// TIA Portal project "ejercicio1" (V15.1)

(* hardware
DEVICE "HMI_1"  KTP700 Basic PN
   slot 0: "HMI_1"  KTP700 Basic PN  6AV2 123-2GB03-0AX0  15.1.0.0
   slot 1: "HMI_RT_1"  KTP700 Basic PN  6AV2 123-2GB03-0AX0  15.1.0.0
   slot 5: "HMI_1.IE_CP_1"  PROFINET Interface  15.0.1.0
      slot 1: "Interfaz PROFINET_1"  PROFINET Interface
         slot 1: "Port_1"  Port
DEVICE "S7-1200 station_1"  S7-1200 Station
   slot 0: "Rack_0"  S7-1200 Rack  Rack  V1.0
   slot 1: "PLC_1"  CPU 1215C AC/DC/Rly  6ES7 215-1BG40-0XB0  V4.2
*)

// ===== PLC "PLC_1"  CPU 1215C AC/DC/Rly =====

VAR_GLOBAL   // PLC tag table "Tabla de variables estándar"
   "q1" AT %M0.0 : Bool;   // estado 1
   "q2" AT %M0.1 : Bool;   // estado 2
   "q3" AT %M0.2 : Bool;   // estado 3
   "q4" AT %M0.3 : Bool;   // estado 4
   "q5" AT %M0.4 : Bool;   // estado 5
   "q6" AT %M0.5 : Bool;   // estado 6
   "MP1" AT %M1.0 : Bool;   // mover der-iz
   "MP2" AT %M1.1 : Bool;   // mover iz-der
   "XV" AT %M1.2 : Bool;   // electrovalvula
   "MC" AT %M1.3 : Bool;   // rodillos
   "MV" AT %M1.4 : Bool;   // ventilador
   "M" AT %M2.0 : Bool;   // boton encendido
   "S1" AT %M2.1 : Bool;   // final de carrera iz
   "S2" AT %M2.2 : Bool;   // final de carrera der
   "S3" AT %M2.3 : Bool;   // detector de coches
   "P" AT %M2.4 : Bool;   // boton paro
END_VAR

ORGANIZATION_BLOCK "Main"   // OB1, LAD, ProgramCycle
TITLE = "Main Program Sweep (Cycle)"
{ S7_Optimized_Access := 'TRUE' }
VERSION : 0.1
   VAR_INPUT
      Initial_Call : Bool;   // Initial call of this OB
      Remanence : Bool;   // =True, if remanent data are available
   END_VAR
BEGIN

REGION Network 1: estado 6: paro
   // si detectamos el boton de paro reseteamos todo y activamos el motor para que regrese a su posicion original
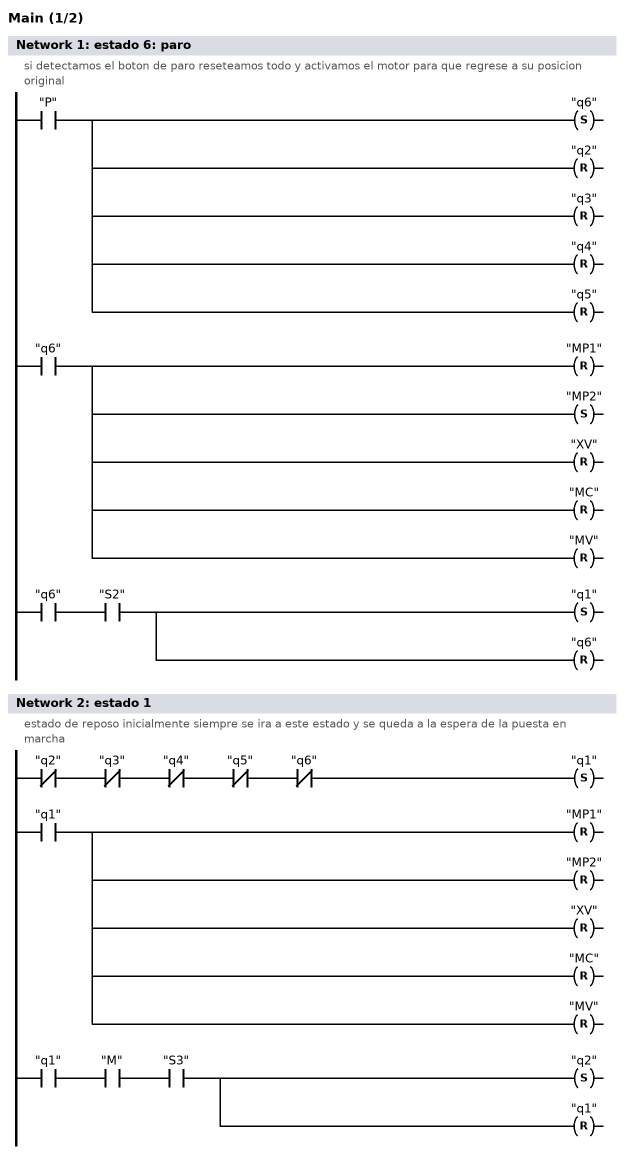
   RUNG wire#powerrail
      Contact( "P" )
      wire#w1
      S_Coil( "q6" )
   END_RUNG
   RUNG wire#w1
      R_Coil( "q2" )
   END_RUNG
   RUNG wire#w1
      R_Coil( "q3" )
   END_RUNG
   RUNG wire#w1
      R_Coil( "q4" )
   END_RUNG
   RUNG wire#w1
      R_Coil( "q5" )
   END_RUNG
   RUNG wire#powerrail
      Contact( "q6" )
      wire#w2
      R_Coil( "MP1" )
   END_RUNG
   RUNG wire#w2
      S_Coil( "MP2" )
   END_RUNG
   RUNG wire#w2
      R_Coil( "XV" )
   END_RUNG
   RUNG wire#w2
      R_Coil( "MC" )
   END_RUNG
   RUNG wire#w2
      R_Coil( "MV" )
   END_RUNG
   RUNG wire#powerrail
      Contact( "q6" )
      Contact( "S2" )
      wire#w3
      S_Coil( "q1" )
   END_RUNG
   RUNG wire#w3
      R_Coil( "q6" )
   END_RUNG
   // the same network as SCL:
   IF "P" THEN
       "q6" := TRUE;
       "q2" := FALSE;
       "q3" := FALSE;
       "q4" := FALSE;
       "q5" := FALSE;
   END_IF;
   IF "q6" THEN
       "MP1" := FALSE;
       "MP2" := TRUE;
       "XV" := FALSE;
       "MC" := FALSE;
       "MV" := FALSE;
   END_IF;
   IF "q6" AND "S2" THEN
       "q1" := TRUE;
       "q6" := FALSE;
   END_IF;
END_REGION

REGION Network 2: estado 1
   // estado de reposo inicialmente siempre se ira a este estado y se queda a la espera de la puesta en marcha
   RUNG wire#powerrail
      I_Contact( "q2" )
      I_Contact( "q3" )
      I_Contact( "q4" )
      I_Contact( "q5" )
      I_Contact( "q6" )
      S_Coil( "q1" )
   END_RUNG
   RUNG wire#powerrail
      Contact( "q1" )
      wire#w1
      R_Coil( "MP1" )
   END_RUNG
   RUNG wire#w1
      R_Coil( "MP2" )
   END_RUNG
   RUNG wire#w1
      R_Coil( "XV" )
   END_RUNG
   RUNG wire#w1
      R_Coil( "MC" )
   END_RUNG
   RUNG wire#w1
      R_Coil( "MV" )
   END_RUNG
   RUNG wire#powerrail
      Contact( "q1" )
      Contact( "M" )
      Contact( "S3" )
      wire#w2
      S_Coil( "q2" )
   END_RUNG
   RUNG wire#w2
      R_Coil( "q1" )
   END_RUNG
   // the same network as SCL:
   IF NOT "q2" AND NOT "q3" AND NOT "q4" AND NOT "q5" AND NOT "q6" THEN "q1" := TRUE; END_IF;
   IF "q1" THEN
       "MP1" := FALSE;
       "MP2" := FALSE;
       "XV" := FALSE;
       "MC" := FALSE;
       "MV" := FALSE;
   END_IF;
   IF "q1" AND "M" AND "S3" THEN
       "q2" := TRUE;
       "q1" := FALSE;
   END_IF;
END_REGION

REGION Network 3: Estado 2
   // ida lavado
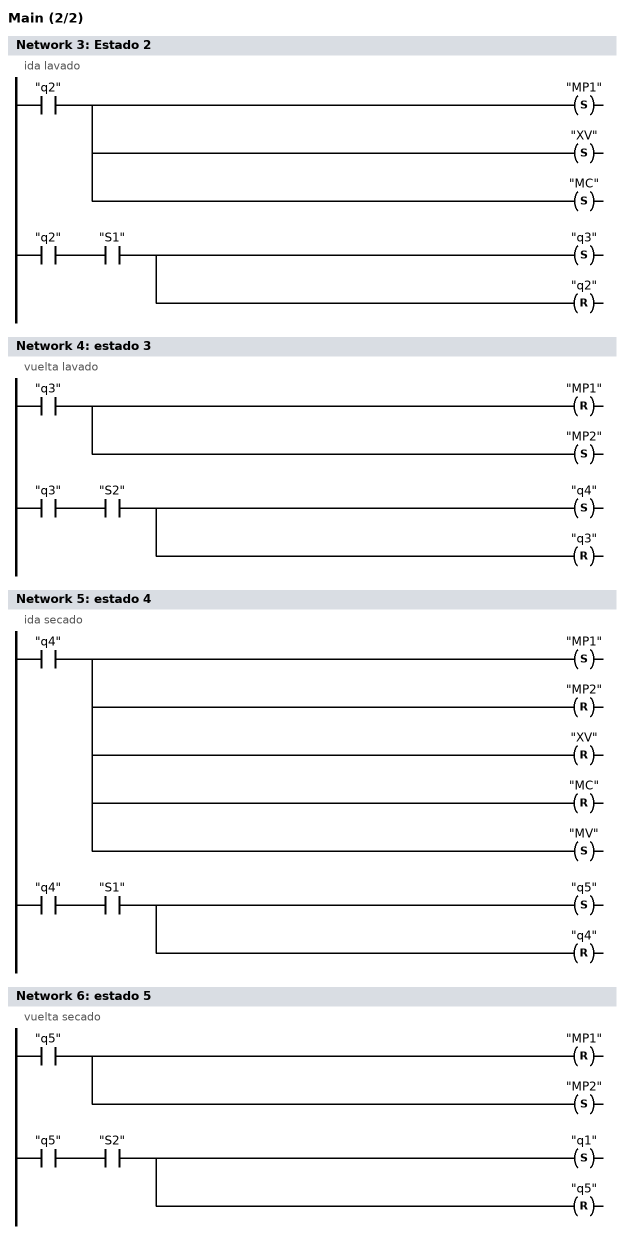
   RUNG wire#powerrail
      Contact( "q2" )
      wire#w1
      S_Coil( "MP1" )
   END_RUNG
   RUNG wire#w1
      S_Coil( "XV" )
   END_RUNG
   RUNG wire#w1
      S_Coil( "MC" )
   END_RUNG
   RUNG wire#powerrail
      Contact( "q2" )
      Contact( "S1" )
      wire#w2
      S_Coil( "q3" )
   END_RUNG
   RUNG wire#w2
      R_Coil( "q2" )
   END_RUNG
   // the same network as SCL:
   IF "q2" THEN
       "MP1" := TRUE;
       "XV" := TRUE;
       "MC" := TRUE;
   END_IF;
   IF "q2" AND "S1" THEN
       "q3" := TRUE;
       "q2" := FALSE;
   END_IF;
END_REGION

REGION Network 4: estado 3
   // vuelta lavado
   RUNG wire#powerrail
      Contact( "q3" )
      wire#w1
      R_Coil( "MP1" )
   END_RUNG
   RUNG wire#w1
      S_Coil( "MP2" )
   END_RUNG
   RUNG wire#powerrail
      Contact( "q3" )
      Contact( "S2" )
      wire#w2
      S_Coil( "q4" )
   END_RUNG
   RUNG wire#w2
      R_Coil( "q3" )
   END_RUNG
   // the same network as SCL:
   IF "q3" THEN
       "MP1" := FALSE;
       "MP2" := TRUE;
   END_IF;
   IF "q3" AND "S2" THEN
       "q4" := TRUE;
       "q3" := FALSE;
   END_IF;
END_REGION

REGION Network 5: estado 4
   // ida secado
   RUNG wire#powerrail
      Contact( "q4" )
      wire#w1
      S_Coil( "MP1" )
   END_RUNG
   RUNG wire#w1
      R_Coil( "MP2" )
   END_RUNG
   RUNG wire#w1
      R_Coil( "XV" )
   END_RUNG
   RUNG wire#w1
      R_Coil( "MC" )
   END_RUNG
   RUNG wire#w1
      S_Coil( "MV" )
   END_RUNG
   RUNG wire#powerrail
      Contact( "q4" )
      Contact( "S1" )
      wire#w2
      S_Coil( "q5" )
   END_RUNG
   RUNG wire#w2
      R_Coil( "q4" )
   END_RUNG
   // the same network as SCL:
   IF "q4" THEN
       "MP1" := TRUE;
       "MP2" := FALSE;
       "XV" := FALSE;
       "MC" := FALSE;
       "MV" := TRUE;
   END_IF;
   IF "q4" AND "S1" THEN
       "q5" := TRUE;
       "q4" := FALSE;
   END_IF;
END_REGION

REGION Network 6: estado 5
   // vuelta secado
   RUNG wire#powerrail
      Contact( "q5" )
      wire#w1
      R_Coil( "MP1" )
   END_RUNG
   RUNG wire#w1
      S_Coil( "MP2" )
   END_RUNG
   RUNG wire#powerrail
      Contact( "q5" )
      Contact( "S2" )
      wire#w2
      S_Coil( "q1" )
   END_RUNG
   RUNG wire#w2
      R_Coil( "q5" )
   END_RUNG
   // the same network as SCL:
   IF "q5" THEN
       "MP1" := FALSE;
       "MP2" := TRUE;
   END_IF;
   IF "q5" AND "S2" THEN
       "q1" := TRUE;
       "q5" := FALSE;
   END_IF;
END_REGION
END_ORGANIZATION_BLOCK

(* ===== HMI "HMI_RT_1" =====
system functions are stored by id; their names below are inferred from use
connection "HMI_Conexión_1": ETHERNET, SMART_S7_1200_OMS

HMI tags "Tabla de variables estándar"
   "Número_imagen_variable" : UInt, internal
   "M" : Bool = PLC M AT %M2.0, 1 s
   "MP1" : Bool = PLC MP1 AT %M1.0, 1 s
   "MP2" : Bool = PLC MP2 AT %M1.1, 1 s
   "XV" : Bool = PLC XV AT %M1.2, 1 s
   "MV" : Bool = PLC MV AT %M1.4, 1 s
   "MC" : Bool = PLC MC AT %M1.3, 1 s
   "q6" : Bool = PLC q6 AT %M0.5, 1 s
   "q1" : Bool = PLC q1 AT %M0.0, 1 s
   "q2" : Bool = PLC q2 AT %M0.1, 1 s
   "q3" : Bool = PLC q3 AT %M0.2, 1 s
   "q4" : Bool = PLC q4 AT %M0.3, 1 s
   "q5" : Bool = PLC q5 AT %M0.4, 1 s
   "S1" : Bool = PLC S1 AT %M2.1, 1 s
   "S2" : Bool = PLC S2 AT %M2.2, 1 s
   "S3" : Bool = PLC S3 AT %M2.3, 1 s
   "P" : Bool = PLC P AT %M2.4, 1 s

text list "Nombre_imagen_lista_texto": 1 'Imagen raíz'

Template "Plantilla_1" 800x480
   Button "Salir" at 714,429 size 71x50; TextOff 'Salir'; PictureOff "ExitRuntime_KTP700_Basic_PN_TR"; PictureOn "ExitRuntime_KTP700_Basic_PN_TR"
      on Release: StopRuntime(0)
   Button "Template_Button" at 614,429 size 71x50; TextOff 'Text'
   Button "Template_Button_1" at 514,429 size 71x50; TextOff 'Text'
   Button "Template_Button_2" at 414,429 size 71x50; TextOff 'Text'
   Button "Template_Button_3" at 314,429 size 71x50; TextOff 'Text'
   Button "Template_Button_4" at 214,429 size 71x50; TextOff 'Text'
   Button "Avisos" at 114,429 size 71x50; TextOff 'Avisos'; PictureOff "AlarmDisplay_KTP700_Basic_PN_TR"; PictureOn "AlarmDisplay_KTP700_Basic_PN_TR"
      on Release: function_ef3f5d25("Ventana de avisos_no_acusado", -1)
   Button "Imagen inicial" at 14,429 size 71x50; TextOff 'Imagen inicial'; PictureOff "NavigateHome_KTP700_Basic_PN_TR"; PictureOn "NavigateHome_KTP700_Basic_PN_TR"
      on Release: ActivateScreen("Imagen raíz", 0)
   SymbolicIOField "Imagen_campo_ES_simbólico" at 93,9 size 600x33; TextOff '0'; TextOn '1'; TextList "Nombre_imagen_lista_texto"
      ProcessValue <- "Número_imagen_variable"
      on Change: ActivateScreenByNumber("Número_imagen_variable", 0)
   DateTimeField "HmiScreenItemData" at 695,25 size 105x25
   DateTimeField "HmiScreenItemData_1" at 695,0 size 105x25
   GraphicView "Logotipo" at 0,0 size 91x51; Picture "Logotipo de HMI_1"

screen "Imagen raíz" 800x480, template "Plantilla_1"
   on GenerateScreen: SetTag("Número_imagen_variable", 1)
   GraphicIOField "PlotLight_Round_G" at 702,60 size 50x50; PictureOn "PilotLight_Round_G_On_256c"; PictureOff "PilotLight_Round_G_Off_256c"
      ProcessValue <- "q1"
   GraphicIOField "PlotLight_Round_R" at 430,60 size 50x50; PictureOn "PilotLight_Round_R_On_256c"; PictureOff "PilotLight_Round_R_Off_256c"
      ProcessValue <- "q6"
   TextField "Campo de texto_1" at 31,137 size 16x23; Text 'Text'
   TextField "Campo de texto_2" at 170,137 size 16x23; Text 'Text'
   TextField "Campo de texto_3" at 638,75 size 60x23; Text 'Espera'
   GraphicIOField "PlotLight_Round_G_1" at 703,132 size 50x50; PictureOff "PilotLight_Round_G_Off_256c"; PictureOn "PilotLight_Round_G_On_256c"
      ProcessValue <- "q2"
   TextField "Campo de texto_4" at 610,147 size 91x23; Text 'Ida lavado'
   GraphicIOField "PlotLight_Round_G_2" at 702,205 size 50x50; PictureOff "PilotLight_Round_G_Off_256c"; PictureOn "PilotLight_Round_G_On_256c"
      ProcessValue <- "q3"
   TextField "Campo de texto_5" at 587,215 size 115x23; Text 'vuelta lavado'
   GraphicIOField "PlotLight_Round_G_3" at 706,274 size 50x50; PictureOn "PilotLight_Round_G_On_256c"; PictureOff "PilotLight_Round_G_Off_256c"
      ProcessValue <- "q4"
   TextField "Campo de texto_6" at 610,287 size 93x23; Text 'Ida secado'
   GraphicIOField "PlotLight_Round_G_4" at 706,347 size 50x50; PictureOff "PilotLight_Round_G_Off_256c"; PictureOn "PilotLight_Round_G_On_256c"
      ProcessValue <- "q5"
   TextField "Campo de texto_7" at 582,358 size 119x23; Text 'Vuelta secado'
   TextField "Campo de texto_8" at 411,109 size 85x23; Text 'Volviendo'
   GraphicIOField "PlotLight_Round_N_Mono_2" at 39,203 size 50x50; PictureOff "PilotLight_Round_N_Off_mono"; PictureOn "PilotLight_Round_N_On_mono"
      ProcessValue <- "MP1"
   TextField "Campo de texto_9" at 44,253 size 40x23; Text 'MP1'
   GraphicIOField "PlotLight_Round_N_Mono_1" at 96,203 size 50x50; PictureOn "PilotLight_Round_N_On_mono"; PictureOff "PilotLight_Round_N_Off_mono"
      ProcessValue <- "MP2"
   TextField "Campo de texto_10" at 101,253 size 40x23; Text 'MP2'
   GraphicIOField "PlotLight_Round_N_Mono_3" at 151,203 size 50x50; PictureOff "PilotLight_Round_N_Off_mono"; PictureOn "PilotLight_Round_N_On_mono"
      ProcessValue <- "XV"
   TextField "Campo de texto_11" at 163,253 size 27x23; Text 'XV'
   GraphicIOField "PlotLight_Round_N_Mono_4" at 205,203 size 50x50; PictureOff "PilotLight_Round_N_Off_mono"; PictureOn "PilotLight_Round_N_On_mono"
      ProcessValue <- "MV"
   TextField "Campo de texto_12" at 215,253 size 30x23; Text 'MV'
   GraphicIOField "PlotLight_Round_N_Mono_5" at 260,203 size 50x50; PictureOn "PilotLight_Round_N_On_mono"; PictureOff "PilotLight_Round_N_Off_mono"
      ProcessValue <- "MC"
   TextField "Campo de texto_13" at 272,253 size 30x23; Text 'MC'
   Button "Botón_1" at 48,332 size 96x32; TextOff 'S1'
      on Press: SetBit("S1")
      Appearance <- "S1"
      on Release: ResetBit("S1")
   Button "Botón_3" at 201,332 size 96x32; TextOff 'S2'
      on Press: SetBit("S2")
      Appearance <- "S2"
      on Release: ResetBit("S2")
   Button "Botón_4" at 355,332 size 96x32; TextOff 'S3'
      on Press: SetBit("S3")
      Appearance <- "S3"
      on Release: ResetBit("S3")
   Button "D1_Pushbutton_Pressed_Off_Green" at 60,60 size 100x66; TextOff 'Text'; PictureOn "Design_1_Button_Green_Pressed_Off"; PictureOff "Design_1_Button_Green_Released_On"
      on Press: SetBit("M")
   Button "D1_Pushbutton_Pressed_Off_Red" at 209,60 size 100x66; TextOff 'Text'; PictureOn "Design_1_Button_Red_Pressed_Off"; PictureOff "Design_1_Button_Red_Released_On"
      on Press: SetBit("P")
      on Release: ResetBit("P")
   TextField "Campo de texto_14" at 63,126 size 88x23; Text 'Encendido'
   TextField "Campo de texto_15" at 234,132 size 43x23; Text 'Paro'
*)